SUBAPPLICATION Uebung_225b_AX (* Dreieck-Sollwertmarker (wie Uebung_225b in test_B, aber mit AR-Adapter-Bausteinen: NumericValue_PHYSA, PositionMarkerFSA, Q_NumericValue_PHYSA) *)
  (* Standard: 61499-2; Description: Copyright (c) 2026 Meisterschulen am Ostbahnhof This program and the accompanying materials are made available under the terms of the Eclipse Public License 2.0 which is available at https://www.eclipse.org/legal/epl-2.0/ SPDX-License-Identifier: EPL-2.0 *)
  (* Version 1.1, 2026-09-06, Franz Höpfinger, Meisterschulen am Ostbahnhof, Enable xScale on Marker_Dreieck *)
  (* Version 1.0, 2026-09-05, Franz Höpfinger, Meisterschulen am Ostbahnhof, adapter variant of Uebung_225b_AX using NumericValue_PHYSA/PositionMarkerFSA/Q_NumericValue_PHYSA *)
  PACKAGE Uebungen;
  IMPORT Uebungen::const::UT::Dreieck::DefaultPool_Dreieck_PositionMarker::Container_PositionMarker;
  IMPORT Uebungen::const::UT::Dreieck::DefaultPool_Dreieck_Numeric::NumberVariable_Sollwert_N;
  IMPORT Uebungen::const::UT::Dreieck::DefaultPool_Dreieck_Numeric::NumberVariable_Istwert_N;
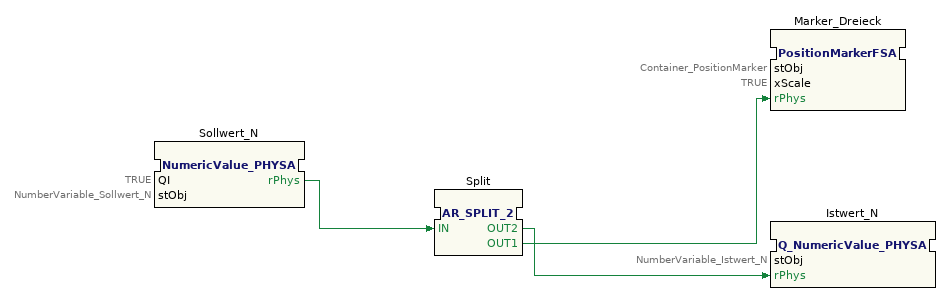
  FBS
    Sollwert_N : isobus::UT::io::NumericValue::NumericValue_PHYSA(QI := TRUE, stObj := NumberVariable_Sollwert_N);
    Split : adapter::events::unidirectional::AR_SPLIT_2;
    Marker_Dreieck : isobus::UT::Q::PositionMarkerFSA(stObj := Container_PositionMarker, xScale := TRUE);
    Istwert_N : isobus::UT::Q::Q_NumericValue_PHYSA(stObj := NumberVariable_Istwert_N);
  END_FBS
  ADAPTER_CONNECTIONS
    Sollwert_N.rPhys TO Split.IN;
    Split.OUT2 TO Istwert_N.rPhys;
    Split.OUT1 TO Marker_Dreieck.rPhys;
  END_CONNECTIONS
END_SUBAPPLICATION
